GLOBALCONSTANTS AID_EX (* External object attribute ids *)
  (* Standard: 61499-1; Description: Copyright (c) 2023 HR Agrartechnik GmbH This program and the accompanying materials are made available under the terms of the Eclipse Public License 2.0 which is available at https://www.eclipse.org/legal/epl-2.0/ SPDX-License-Identifier: EPL-2.0 *)
  (* Version 1.0, 2026-06-20, Franz Höpfinger, HR Agrartechnik GmbH *)
  PACKAGE isobus::UT::Q::const::AID;
  VAR_GLOBAL CONSTANT
    OPTIONS : USINT := USINT#1; (* 1: AID_EX_OPTIONS - Bitmask: Bit 0 = Enabled (allows referenced NAME WS to reference listed *)
    NAME_0 : USINT := USINT#2; (* 2: AID_EX_NAME_0 *)
    NAME_1 : USINT := USINT#3; (* 3: AID_EX_NAME_1 *)
  END_VAR
END_GLOBALCONSTANTS
